INTERFACE  I_PersistantEventStorage

METHOD M_StoreEvent
VAR_INPUT
	stEvent : ST_Event;
END_VAR
END_METHOD

END_INTERFACE

(* stored: Version 1.1.0.1
   Itf I_PersistantEventStorage: Id {b1c6bde6-fb2a-4538-8e38-a39d4d9696ff}
   Method M_StoreEvent: Id {3e3c3203-7574-46d4-8247-85fe611e6148} *)
